DATA_BLOCK "$NAME"
TITLE = $TITLE
VERSION : $VERSION
$RETAIN
    STRUCT
        @PARAMETERS[$NAME : $TYPE; //$COMMENT]
    END_STRUCT ;
BEGIN
    @PARAMETERS_VALUES[$NAME := $VALUE;]
END_DATA_BLOCK